(* IEC 61131-3 sources: volt/packages/volt-lsp-iec/test-corpus/lenze-mid/Device/Plc Logic/Application/Library Manager/CAA File, 66 files *)

(* ---- ATTRIB.dut ---- *)
TYPE ATTRIB :
(
	ARCHIVE := 0,
	HIDDEN,
	NORMAL,
	READONLY
);
END_TYPE

(* ---- ERROR.dut ---- *)
TYPE ERROR :
(
	NO_ERROR := 0,
	FIRST_ERROR := 5100,
	TIME_OUT,
	ABORT,
	HANDLE_INVALID,
	NOT_EXIST,
	EXIST,
	NO_MORE_ENTRIES,
	NOT_EMPTY,
	READ_ONLY_CAA,
	WRONG_PARAMETER,
	ERROR_UNKNOWN,
	WRITE_INCOMPLETE,
	FILE_NOT_IMPLEMENTED,
	ASM_CREATEJOB_FAILED,
	FILE_OPERATION_DENIED,
	FIRST_MF := 5150,
	LAST_ERROR := 5199
);
END_TYPE

(* ---- FILE_CLOSE_PARAMS.dut ---- *)
TYPE FILE_CLOSE_PARAMS :
STRUCT
	HFILE : CAA.HANDLE;
END_STRUCT
END_TYPE

(* ---- FILE_COPY_PARAMS.dut ---- *)
TYPE FILE_COPY_PARAMS :
STRUCT
	SFILENAMEDEST : CAA.FILENAME;
	SFILENAMESOURCE : CAA.FILENAME;
	XOVERWRITE : BOOL;
	ABYDUMMY : ARRAY [0..2] OF BYTE;
	SZSIZE : CAA.SIZE;
END_STRUCT
END_TYPE

(* ---- FILE_DELETE_PARAMS.dut ---- *)
TYPE FILE_DELETE_PARAMS :
STRUCT
	SFILENAME : CAA.FILENAME;
END_STRUCT
END_TYPE

(* ---- FILE_DIR_ENTRY.dut ---- *)
TYPE FILE_DIR_ENTRY :
STRUCT
	SENTRY : CAA.FILENAME;
	SZSIZE : CAA.SIZE;
	XDIRECTORY : BOOL;
	XEXCLUSIVE : BOOL;
	DTLASTMODIFICATION : DATE_AND_TIME;
END_STRUCT
END_TYPE

(* ---- FILE_DIRCLOSE_PARAMS.dut ---- *)
TYPE FILE_DIRCLOSE_PARAMS :
STRUCT
	HDIR : CAA.HANDLE;
END_STRUCT
END_TYPE

(* ---- FILE_DIRCOPY_PARAMS.dut ---- *)
TYPE FILE_DIRCOPY_PARAMS :
STRUCT
	SDIRNAMEDEST : CAA.FILENAME;
	SDIRNAMESOURCE : CAA.FILENAME;
	XRECURSIVE : BOOL;
	XOVERWRITE : BOOL;
END_STRUCT
END_TYPE

(* ---- FILE_DIRCREATE_PARAMS.dut ---- *)
TYPE FILE_DIRCREATE_PARAMS :
STRUCT
	SDIRNAME : CAA.FILENAME;
	XPARENT : BOOL;
END_STRUCT
END_TYPE

(* ---- FILE_DIRLIST_PARAMS.dut ---- *)
TYPE FILE_DIRLIST_PARAMS :
STRUCT
	HDIR : CAA.HANDLE;
	DEDIRENTRY : FILE_DIR_ENTRY;
END_STRUCT
END_TYPE

(* ---- FILE_DIROPEN_PARAMS.dut ---- *)
TYPE FILE_DIROPEN_PARAMS :
STRUCT
	SDIRNAME : CAA.FILENAME;
	HDIR : CAA.HANDLE;
END_STRUCT
END_TYPE

(* ---- FILE_DIRREMOVE_PARAMS.dut ---- *)
TYPE FILE_DIRREMOVE_PARAMS :
STRUCT
	SDIRNAME : CAA.FILENAME;
	XRECURSIVE : BOOL;
END_STRUCT
END_TYPE

(* ---- FILE_DIRRENAME_PARAMS.dut ---- *)
TYPE FILE_DIRRENAME_PARAMS :
STRUCT
	SDIRNAMEOLD : CAA.FILENAME;
	SDIRNAMENEW : CAA.FILENAME;
END_STRUCT
END_TYPE

(* ---- FILE_EOF_PARAMS.dut ---- *)
TYPE FILE_EOF_PARAMS :
STRUCT
	HFILE : CAA.HANDLE;
	XEOF : BOOL;
END_STRUCT
END_TYPE

(* ---- FILE_FLUSH_PARAMS.dut ---- *)
TYPE FILE_FLUSH_PARAMS :
STRUCT
	HFILE : CAA.HANDLE;
END_STRUCT
END_TYPE

(* ---- FILE_GETAT_PARAMS.dut ---- *)
TYPE FILE_GETAT_PARAMS :
STRUCT
	HFILE : CAA.HANDLE;
	EFILEATTRIB : ATTRIB;
END_STRUCT
END_TYPE

(* ---- FILE_GETPOS_PARAMS.dut ---- *)
TYPE FILE_GETPOS_PARAMS :
STRUCT
	HFILE : CAA.HANDLE;
	UDIPOS : __UXINT;
END_STRUCT
END_TYPE

(* ---- FILE_GETROOT_PARAMS.dut ---- *)
TYPE FILE_GETROOT_PARAMS :
STRUCT
	SFILENAME : CAA.FILENAME;
END_STRUCT
END_TYPE

(* ---- FILE_GETSIZE_PARAMS.dut ---- *)
TYPE FILE_GETSIZE_PARAMS :
STRUCT
	SFILENAME : CAA.FILENAME;
	SZSIZE : CAA.SIZE;
END_STRUCT
END_TYPE

(* ---- FILE_GETTIME_PARAMS.dut ---- *)
TYPE FILE_GETTIME_PARAMS :
STRUCT
	SFILENAME : CAA.FILENAME;
	DTLASTMODIFICATION : DATE_AND_TIME;
END_STRUCT
END_TYPE

(* ---- FILE_OPEN_PARAMS.dut ---- *)
TYPE FILE_OPEN_PARAMS :
STRUCT
	SFILENAME : CAA.FILENAME;
	EFILEMODE : MODE;
	XEXCLUSIVE : BOOL;
	BYDUMMY : BOOL;
	HFILE : CAA.HANDLE;
END_STRUCT
END_TYPE

(* ---- FILE_READ_PARAMS.dut ---- *)
TYPE FILE_READ_PARAMS :
STRUCT
	HFILE : CAA.HANDLE;
	PBUFFER : CAA.PVOID;
	SZBUFFER : CAA.SIZE;
	SZSIZE : CAA.SIZE;
END_STRUCT
END_TYPE

(* ---- FILE_RENAME_PARAMS.dut ---- *)
TYPE FILE_RENAME_PARAMS :
STRUCT
	SFILENAMEOLD : CAA.FILENAME;
	SFILENAMENEW : CAA.FILENAME;
END_STRUCT
END_TYPE

(* ---- FILE_SETAT_PARAMS.dut ---- *)
TYPE FILE_SETAT_PARAMS :
STRUCT
	HFILE : CAA.HANDLE;
	EFILEATTRIB : ATTRIB;
END_STRUCT
END_TYPE

(* ---- FILE_SETPOS_PARAMS.dut ---- *)
TYPE FILE_SETPOS_PARAMS :
STRUCT
	HFILE : CAA.HANDLE;
	UDIPOS : __UXINT;
END_STRUCT
END_TYPE

(* ---- FILE_SETROOT_PARAMS.dut ---- *)
TYPE FILE_SETROOT_PARAMS :
STRUCT
	SFILENAME : CAA.FILENAME;
END_STRUCT
END_TYPE

(* ---- FILE_WRITE_PARAMS.dut ---- *)
TYPE FILE_WRITE_PARAMS :
STRUCT
	HFILE : CAA.HANDLE;
	PBUFFER : CAA.PVOID;
	SZSIZE : CAA.SIZE;
END_STRUCT
END_TYPE

(* ---- MODE.dut ---- *)
TYPE MODE :
(
	MWRITE := 0,
	MREAD,
	MRDWR,
	MAPPD,
	MREADPLUS,
	MWRITEPLUS,
	MAPPENDPLUS
);
END_TYPE

(* ---- CAA_ASM_CONSTANTS.gvl ---- *)
VAR_GLOBAL
	OPEN_JOB_ID : UDINT := 16#10001;
	CLOSE_JOB_ID : UDINT := 16#10002;
	COPY_JOB_ID : UDINT := 16#10003;
	DELETE_JOB_ID : UDINT := 16#10004;
	EOF_JOB_ID : UDINT := 16#10005;
	GETPOS_JOB_ID : UDINT := 16#10006;
	GETSIZE_JOB_ID : UDINT := 16#10007;
	GETTIME_JOB_ID : UDINT := 16#10008;
	READ_JOB_ID : UDINT := 16#10009;
	RENAME_JOB_ID : UDINT := 16#1000A;
	SETATTRIBUTE_JOB_ID : UDINT := 16#1000B;
	SETPOS_JOB_ID : UDINT := 16#1000C;
	WRITE_JOB_ID : UDINT := 16#1000D;
	GETROOT_JOB_ID : UDINT := 16#1000E;
	SETROOT_JOB_ID : UDINT := 16#1000F;
	DIRCLOSE_JOB_ID : UDINT := 16#10010;
	DIRCREATE_JOB_ID : UDINT := 16#10011;
	DIRLIST_JOB_ID : UDINT := 16#10012;
	DIROPEN_JOB_ID : UDINT := 16#10013;
	DIRREMOVE_JOB_ID : UDINT := 16#10014;
	DIRRENAME_JOB_ID : UDINT := 16#10015;
	FLUSH_JOB_ID : UDINT := 16#10016;
	GETATTRIBUTE_JOB_ID : UDINT := 16#10017;
	DIRCOPY_JOB_ID : UDINT := 16#10018;
END_VAR

(* ---- CAA_GLOBALE_CONSTANTS.gvl ---- *)
VAR_GLOBAL
	GC_PDIRNAME : WORD := 1;
	GC_PRENAME : WORD := 2;
	GC_PCOPY : WORD := 3;
	GC_PSETATTRIBUTE : WORD := 4;
	GC_PFILENAME83 : WORD := 100;
	GC_PCAPITALLETTERS : WORD := 101;
	GC_PABSOLUTEPATH : WORD := 200;
	GC_PDRIVELETTER : WORD := 201;
	GC_PNETWORKDRIVES : WORD := 300;
END_VAR

(* ---- EXAMPLES.gvl ---- *)
VAR_GLOBAL
	IDUMMYFORLIBDOCUCAAFILE : INT := 99;
END_VAR

(* ---- RSHANDLING.gvl ---- *)
VAR_GLOBAL
	G_FILECLASS : FileClass;
	G_DIRCLASS : DirClass;
END_VAR

(* ---- VERSIONCONSTANTS.gvl ---- *)
VAR_GLOBAL
	GC_BYVERSION : BYTE := 1;
	GC_BYVERSION_1 : BYTE := 0;
END_VAR

(* ---- _CLOSE.pou ---- *)
FUNCTION _CLOSE : ERROR
VAR_INPUT
	HFILE : CAA.HANDLE;
END_VAR
END_FUNCTION

(* ---- _DIRCLOSE.pou ---- *)
FUNCTION _DIRCLOSE : ERROR
VAR_INPUT
	HDIR : CAA.HANDLE;
END_VAR
END_FUNCTION

(* ---- GETLIBVERSION.pou ---- *)
FUNCTION GETLIBVERSION : VERSION
END_FUNCTION

(* ---- GETLIBVERSIONNUMBER.pou ---- *)
FUNCTION GETLIBVERSIONNUMBER : DWORD
END_FUNCTION

(* ---- GETPROPERTY.pou ---- *)
FUNCTION GETPROPERTY : DWORD
VAR_INPUT
	WPROPERTY : WORD;
END_VAR
END_FUNCTION

(* ---- GETSUPPLIERVERSION.pou ---- *)
FUNCTION GETSUPPLIERVERSION : WORD
VAR_INPUT
	XDUMMY : BOOL;
END_VAR
END_FUNCTION

(* ---- ISLIBRELEASED.pou ---- *)
FUNCTION ISLIBRELEASED : BOOL
END_FUNCTION

(* ---- CLOSE.pou ---- *)
FUNCTION_BLOCK CLOSE EXTENDS ETrig
VAR_INPUT
	HFILE : CAA.HANDLE;
END_VAR
VAR_OUTPUT
	EERROR : ERROR;
END_VAR
VAR
	HJOB : CAA.HANDLE;
	PFILECLOSEPARAMS : POINTER TO FILE_CLOSE_PARAMS;
	STATEJOB : ASM.STATE;
	FILECLOSEPARAMS : FILE_CLOSE_PARAMS;
END_VAR
END_FUNCTION_BLOCK

METHOD PRVABORT : BOOL
END_METHOD

METHOD PRVCYCLICACTION : BOOL
END_METHOD

METHOD PRVRESETOUTPUTS : BOOL
END_METHOD

METHOD PRVSTART : BOOL
END_METHOD

(* ---- COPY.pou ---- *)
FUNCTION_BLOCK COPY EXTENDS ETrigToA
VAR_INPUT
	SFILENAMEDEST : CAA.FILENAME;
	SFILENAMESOURCE : CAA.FILENAME;
	XOVERWRITE : BOOL := TRUE;
END_VAR
VAR_OUTPUT
	EERROR : ERROR;
	SZSIZE : CAA.SIZE;
END_VAR
VAR
	HJOB : CAA.HANDLE;
	PFILECOPYPARAMS : POINTER TO FILE_COPY_PARAMS;
	STATEJOB : ASM.STATE;
	FILECOPYPARAMS : FILE_COPY_PARAMS;
END_VAR
END_FUNCTION_BLOCK

METHOD PRVABORT : BOOL
END_METHOD

METHOD PRVCYCLICACTION : BOOL
END_METHOD

METHOD PRVRESETOUTPUTS : BOOL
END_METHOD

METHOD PRVSTART : BOOL
END_METHOD

(* ---- DELETE.pou ---- *)
FUNCTION_BLOCK DELETE EXTENDS ETrig
VAR_INPUT
	SFILENAME : CAA.FILENAME;
END_VAR
VAR_OUTPUT
	EERROR : ERROR;
END_VAR
VAR
	HJOB : CAA.HANDLE;
	PFILEDELETEPARAMS : POINTER TO FILE_DELETE_PARAMS;
	STATEJOB : ASM.STATE;
	FILEDELETEPARAMS : FILE_DELETE_PARAMS;
END_VAR
END_FUNCTION_BLOCK

METHOD PRVABORT : BOOL
END_METHOD

METHOD PRVCYCLICACTION : BOOL
END_METHOD

METHOD PRVRESETOUTPUTS : BOOL
END_METHOD

METHOD PRVSTART : BOOL
END_METHOD

(* ---- DIRCLASS.pou ---- *)
FUNCTION_BLOCK DIRCLASS EXTENDS RSMClass
END_FUNCTION_BLOCK

METHOD CLOSE : RSM.ERROR
VAR_INPUT
	HHANDLE : CAA.HANDLE;
END_VAR
END_METHOD

(* ---- DIRCLOSE.pou ---- *)
FUNCTION_BLOCK DIRCLOSE EXTENDS ETrig
VAR_INPUT
	HDIR : CAA.HANDLE;
END_VAR
VAR_OUTPUT
	EERROR : ERROR;
END_VAR
VAR
	HJOB : CAA.HANDLE;
	PDIRCLOSEPARAMS : POINTER TO FILE_DIRCLOSE_PARAMS;
	STATEJOB : ASM.STATE;
	DIRCLOSEPARAMS : FILE_DIRCLOSE_PARAMS;
END_VAR
END_FUNCTION_BLOCK

METHOD PRVSTART : BOOL
END_METHOD

METHOD PRVCYCLICACTION : BOOL
END_METHOD

METHOD PRVRESETOUTPUTS : BOOL
END_METHOD

METHOD PRVABORT : BOOL
END_METHOD

(* ---- DIRCOPY.pou ---- *)
FUNCTION_BLOCK DIRCOPY EXTENDS ETrig
VAR_INPUT
	SDIRNAMEDEST : CAA.FILENAME;
	SDIRNAMESOURCE : CAA.FILENAME;
	XRECURSIVE : BOOL;
	XOVERWRITE : BOOL;
END_VAR
VAR_OUTPUT
	EERROR : ERROR;
END_VAR
VAR
	HJOB : CAA.HANDLE;
	PDIRCOPYPARAMS : POINTER TO FILE_DIRCOPY_PARAMS;
	STATEJOB : ASM.STATE;
	DIRCOPYPARAMS : FILE_DIRCOPY_PARAMS;
END_VAR
END_FUNCTION_BLOCK

METHOD PRVCYCLICACTION : BOOL
END_METHOD

METHOD PRVRESETOUTPUTS : BOOL
END_METHOD

METHOD PRVABORT : BOOL
END_METHOD

METHOD PRVSTART : BOOL
END_METHOD

(* ---- DIRCREATE.pou ---- *)
FUNCTION_BLOCK DIRCREATE EXTENDS ETrig
VAR_INPUT
	SDIRNAME : CAA.FILENAME;
	XPARENT : BOOL;
END_VAR
VAR_OUTPUT
	EERROR : ERROR;
END_VAR
VAR
	HJOB : CAA.HANDLE;
	PDIRCREATEPARAMS : POINTER TO FILE_DIRCREATE_PARAMS;
	STATEJOB : ASM.STATE;
	DIRCREATEPARAMS : FILE_DIRCREATE_PARAMS;
END_VAR
END_FUNCTION_BLOCK

METHOD PRVSTART : BOOL
END_METHOD

METHOD PRVCYCLICACTION : BOOL
END_METHOD

METHOD PRVRESETOUTPUTS : BOOL
END_METHOD

METHOD PRVABORT : BOOL
END_METHOD

(* ---- DIRLIST.pou ---- *)
FUNCTION_BLOCK DIRLIST EXTENDS ETrig
VAR_INPUT
	HDIR : CAA.HANDLE;
END_VAR
VAR_OUTPUT
	EERROR : ERROR;
	DEDIRENTRY : FILE_DIR_ENTRY;
END_VAR
VAR
	HJOB : CAA.HANDLE;
	PDIRLISTPARAMS : POINTER TO FILE_DIRLIST_PARAMS;
	STATEJOB : ASM.STATE;
	DIRLISTPARAMS : FILE_DIRLIST_PARAMS;
END_VAR
END_FUNCTION_BLOCK

METHOD PRVCYCLICACTION : BOOL
END_METHOD

METHOD PRVRESETOUTPUTS : BOOL
END_METHOD

METHOD PRVABORT : BOOL
END_METHOD

METHOD PRVSTART : BOOL
END_METHOD

(* ---- DIROPEN.pou ---- *)
FUNCTION_BLOCK DIROPEN EXTENDS ETrig
VAR_INPUT
	SDIRNAME : CAA.FILENAME;
END_VAR
VAR_OUTPUT
	EERROR : ERROR;
	HDIR : CAA.HANDLE;
END_VAR
VAR
	SCOPYDIRNAME : CAA.FILENAME;
	HJOB : CAA.HANDLE;
	PDIROPENPARAMS : POINTER TO FILE_DIROPEN_PARAMS;
	STATEJOB : ASM.STATE;
	DIROPENPARAMS : FILE_DIROPEN_PARAMS;
END_VAR
END_FUNCTION_BLOCK

METHOD PRVCYCLICACTION : BOOL
END_METHOD

METHOD PRVRESETOUTPUTS : BOOL
END_METHOD

METHOD PRVABORT : BOOL
END_METHOD

METHOD PRVSTART : BOOL
END_METHOD

(* ---- DIRREMOVE.pou ---- *)
FUNCTION_BLOCK DIRREMOVE EXTENDS ETrigToA
VAR_INPUT
	SDIRNAME : CAA.FILENAME;
	XRECURSIVE : BOOL;
END_VAR
VAR_OUTPUT
	EERROR : ERROR;
END_VAR
VAR
	HJOB : CAA.HANDLE;
	PDIRREMOVEPARAMS : POINTER TO FILE_DIRREMOVE_PARAMS;
	STATEJOB : ASM.STATE;
	DIRREMOVEPARAMS : FILE_DIRREMOVE_PARAMS;
END_VAR
END_FUNCTION_BLOCK

METHOD PRVRESETOUTPUTS : BOOL
END_METHOD

METHOD PRVABORT : BOOL
END_METHOD

METHOD PRVSTART : BOOL
END_METHOD

METHOD PRVCYCLICACTION : BOOL
END_METHOD

(* ---- DIRRENAME.pou ---- *)
FUNCTION_BLOCK DIRRENAME EXTENDS ETrig
VAR_INPUT
	SDIRNAMEOLD : CAA.FILENAME;
	SDIRNAMENEW : CAA.FILENAME;
END_VAR
VAR_OUTPUT
	EERROR : ERROR;
END_VAR
VAR
	HJOB : CAA.HANDLE;
	PDIRRENAMEPARAMS : POINTER TO FILE_DIRRENAME_PARAMS;
	STATEJOB : ASM.STATE;
	DIRRENAMEPARAMS : FILE_DIRRENAME_PARAMS;
END_VAR
END_FUNCTION_BLOCK

METHOD PRVRESETOUTPUTS : BOOL
END_METHOD

METHOD PRVABORT : BOOL
END_METHOD

METHOD PRVSTART : BOOL
END_METHOD

METHOD PRVCYCLICACTION : BOOL
END_METHOD

(* ---- EOF.pou ---- *)
FUNCTION_BLOCK EOF EXTENDS ETrig
VAR_INPUT
	HFILE : CAA.HANDLE;
END_VAR
VAR_OUTPUT
	EERROR : ERROR;
	XEOF : BOOL;
END_VAR
VAR
	HJOB : CAA.HANDLE;
	PEOFPARAMS : POINTER TO FILE_EOF_PARAMS;
	STATEJOB : ASM.STATE;
	EOFPARAMS : FILE_EOF_PARAMS;
END_VAR
END_FUNCTION_BLOCK

METHOD PRVABORT : BOOL
END_METHOD

METHOD PRVCYCLICACTION : BOOL
END_METHOD

METHOD PRVRESETOUTPUTS : BOOL
END_METHOD

METHOD PRVSTART : BOOL
END_METHOD

(* ---- FILECLASS.pou ---- *)
FUNCTION_BLOCK FILECLASS EXTENDS RSMClass
END_FUNCTION_BLOCK

METHOD CLOSE : RSM.ERROR
VAR_INPUT
	HHANDLE : CAA.HANDLE;
END_VAR
END_METHOD

(* ---- FLUSH.pou ---- *)
FUNCTION_BLOCK FLUSH EXTENDS ETrig
VAR_INPUT
	HFILE : CAA.HANDLE;
END_VAR
VAR_OUTPUT
	EERROR : ERROR;
END_VAR
VAR
	HJOB : CAA.HANDLE;
	PFLUSHPARAMS : POINTER TO FILE_FLUSH_PARAMS;
	STATEJOB : ASM.STATE;
	FLUSHPARAMS : FILE_FLUSH_PARAMS;
END_VAR
END_FUNCTION_BLOCK

METHOD PRVABORT : BOOL
END_METHOD

METHOD PRVCYCLICACTION : BOOL
END_METHOD

METHOD PRVRESETOUTPUTS : BOOL
END_METHOD

METHOD PRVSTART : BOOL
END_METHOD

(* ---- GETATTRIBUTE.pou ---- *)
FUNCTION_BLOCK GETATTRIBUTE EXTENDS ETrig
VAR_INPUT
	HFILE : CAA.HANDLE;
END_VAR
VAR_OUTPUT
	EERROR : ERROR;
	EFILEATTRIB : ATTRIB;
END_VAR
VAR
	HJOB : CAA.HANDLE;
	PGETATPARAMS : POINTER TO FILE_GETAT_PARAMS;
	STATEJOB : ASM.STATE;
	GETATPARAMS : FILE_GETAT_PARAMS;
END_VAR
END_FUNCTION_BLOCK

METHOD PRVABORT : BOOL
END_METHOD

METHOD PRVCYCLICACTION : BOOL
END_METHOD

METHOD PRVRESETOUTPUTS : BOOL
END_METHOD

METHOD PRVSTART : BOOL
END_METHOD

(* ---- GETPOS.pou ---- *)
FUNCTION_BLOCK GETPOS EXTENDS ETrig
VAR_INPUT
	HFILE : CAA.HANDLE;
END_VAR
VAR_OUTPUT
	EERROR : ERROR;
	UDIPOS : __UXINT;
END_VAR
VAR
	HJOB : CAA.HANDLE;
	PGETPOSPARAMS : POINTER TO FILE_GETPOS_PARAMS;
	STATEJOB : ASM.STATE;
	GETPOSPARAMS : FILE_GETPOS_PARAMS;
END_VAR
END_FUNCTION_BLOCK

METHOD PRVABORT : BOOL
END_METHOD

METHOD PRVCYCLICACTION : BOOL
END_METHOD

METHOD PRVRESETOUTPUTS : BOOL
END_METHOD

METHOD PRVSTART : BOOL
END_METHOD

(* ---- GETROOT.pou ---- *)
FUNCTION_BLOCK GETROOT EXTENDS ETrig
VAR_OUTPUT
	EERROR : ERROR;
	SFILENAME : CAA.FILENAME;
END_VAR
VAR
	HJOB : CAA.HANDLE;
	PGETROOTPARAMS : POINTER TO FILE_GETROOT_PARAMS;
	STATEJOB : ASM.STATE;
	GETROOTPARAMS : FILE_GETROOT_PARAMS;
END_VAR
END_FUNCTION_BLOCK

METHOD PRVCYCLICACTION : BOOL
END_METHOD

METHOD PRVRESETOUTPUTS : BOOL
END_METHOD

METHOD PRVABORT : BOOL
END_METHOD

METHOD PRVSTART : BOOL
END_METHOD

(* ---- GETSIZE.pou ---- *)
FUNCTION_BLOCK GETSIZE EXTENDS ETrig
VAR_INPUT
	SFILENAME : CAA.FILENAME;
END_VAR
VAR_OUTPUT
	EERROR : ERROR;
	SZSIZE : CAA.SIZE;
END_VAR
VAR
	HJOB : CAA.HANDLE;
	PGETSIZEPARAMS : POINTER TO FILE_GETSIZE_PARAMS;
	STATEJOB : ASM.STATE;
	GETSIZEPARAMS : FILE_GETSIZE_PARAMS;
END_VAR
END_FUNCTION_BLOCK

METHOD PRVABORT : BOOL
END_METHOD

METHOD PRVCYCLICACTION : BOOL
END_METHOD

METHOD PRVRESETOUTPUTS : BOOL
END_METHOD

METHOD PRVSTART : BOOL
END_METHOD

(* ---- GETTIME.pou ---- *)
FUNCTION_BLOCK GETTIME EXTENDS ETrig
VAR_INPUT
	SFILENAME : CAA.FILENAME;
END_VAR
VAR_OUTPUT
	EERROR : ERROR;
	DTLASTMODIFICATION : DATE_AND_TIME;
END_VAR
VAR
	HJOB : CAA.HANDLE;
	PGETTIMEPARAMS : POINTER TO FILE_GETTIME_PARAMS;
	STATEJOB : ASM.STATE;
	GETTIMEPARAMS : FILE_GETTIME_PARAMS;
END_VAR
END_FUNCTION_BLOCK

METHOD PRVABORT : BOOL
END_METHOD

METHOD PRVCYCLICACTION : BOOL
END_METHOD

METHOD PRVRESETOUTPUTS : BOOL
END_METHOD

METHOD PRVSTART : BOOL
END_METHOD

(* ---- OPEN.pou ---- *)
FUNCTION_BLOCK OPEN EXTENDS ETrig
VAR_INPUT
	SFILENAME : CAA.FILENAME;
	EFILEMODE : MODE;
	XEXCLUSIVE : BOOL;
END_VAR
VAR_OUTPUT
	EERROR : ERROR;
	HFILE : CAA.HANDLE;
END_VAR
VAR
	HJOB : CAA.HANDLE;
	PFILEOPENPARAMS : POINTER TO FILE_OPEN_PARAMS;
	STATEJOB : ASM.STATE;
	FILEOPENPARAMS : FILE_OPEN_PARAMS;
END_VAR
END_FUNCTION_BLOCK

METHOD PRVABORT : BOOL
END_METHOD

METHOD PRVCYCLICACTION : BOOL
END_METHOD

METHOD PRVRESETOUTPUTS : BOOL
END_METHOD

METHOD PRVSTART : BOOL
END_METHOD

(* ---- READ.pou ---- *)
FUNCTION_BLOCK READ EXTENDS ETrigToA
VAR_INPUT
	HFILE : CAA.HANDLE;
	PBUFFER : CAA.PVOID;
	SZBUFFER : CAA.SIZE;
END_VAR
VAR_OUTPUT
	EERROR : ERROR;
	SZSIZE : CAA.SIZE;
END_VAR
VAR
	HJOB : CAA.HANDLE;
	PREADPARAMS : POINTER TO FILE_READ_PARAMS;
	STATEJOB : ASM.STATE;
	READPARAMS : FILE_READ_PARAMS;
END_VAR
END_FUNCTION_BLOCK

METHOD PRVABORT : BOOL
END_METHOD

METHOD PRVCYCLICACTION : BOOL
END_METHOD

METHOD PRVRESETOUTPUTS : BOOL
END_METHOD

METHOD PRVSTART : BOOL
END_METHOD

(* ---- RENAME.pou ---- *)
FUNCTION_BLOCK RENAME EXTENDS ETrig
VAR_INPUT
	SFILENAMEOLD : CAA.FILENAME;
	SFILENAMENEW : CAA.FILENAME;
END_VAR
VAR_OUTPUT
	EERROR : ERROR;
END_VAR
VAR
	HJOB : CAA.HANDLE;
	PRENAMEPARAMS : POINTER TO FILE_RENAME_PARAMS;
	STATEJOB : ASM.STATE;
	RENAMEPARAMS : FILE_RENAME_PARAMS;
END_VAR
END_FUNCTION_BLOCK

METHOD PRVABORT : BOOL
END_METHOD

METHOD PRVCYCLICACTION : BOOL
END_METHOD

METHOD PRVRESETOUTPUTS : BOOL
END_METHOD

METHOD PRVSTART : BOOL
END_METHOD

(* ---- SETATTRIBUTE.pou ---- *)
FUNCTION_BLOCK SETATTRIBUTE EXTENDS ETrig
VAR_INPUT
	HFILE : CAA.HANDLE;
	EFILEATTRIB : ATTRIB;
END_VAR
VAR_OUTPUT
	EERROR : ERROR;
END_VAR
VAR
	HJOB : CAA.HANDLE;
	PSETATPARAMS : POINTER TO FILE_SETAT_PARAMS;
	STATEJOB : ASM.STATE;
	SETATPARAMS : FILE_SETAT_PARAMS;
END_VAR
END_FUNCTION_BLOCK

METHOD PRVABORT : BOOL
END_METHOD

METHOD PRVCYCLICACTION : BOOL
END_METHOD

METHOD PRVRESETOUTPUTS : BOOL
END_METHOD

METHOD PRVSTART : BOOL
END_METHOD

(* ---- SETPOS.pou ---- *)
FUNCTION_BLOCK SETPOS EXTENDS ETrig
VAR_INPUT
	HFILE : CAA.HANDLE;
	UDIPOS : __UXINT;
END_VAR
VAR_OUTPUT
	EERROR : ERROR;
END_VAR
VAR
	HJOB : CAA.HANDLE;
	PSETPOSPARAMS : POINTER TO FILE_SETPOS_PARAMS;
	STATEJOB : ASM.STATE;
	SETPOSPARAMS : FILE_SETPOS_PARAMS;
END_VAR
END_FUNCTION_BLOCK

METHOD PRVABORT : BOOL
END_METHOD

METHOD PRVCYCLICACTION : BOOL
END_METHOD

METHOD PRVRESETOUTPUTS : BOOL
END_METHOD

METHOD PRVSTART : BOOL
END_METHOD

(* ---- SETROOT.pou ---- *)
FUNCTION_BLOCK SETROOT EXTENDS ETrig
VAR_INPUT
	SFILENAME : CAA.FILENAME;
END_VAR
VAR_OUTPUT
	EERROR : ERROR;
END_VAR
VAR
	HJOB : CAA.HANDLE;
	PSETROOTPARAMS : POINTER TO FILE_SETROOT_PARAMS;
	STATEJOB : ASM.STATE;
	SETROOTPARAMS : FILE_SETROOT_PARAMS;
END_VAR
END_FUNCTION_BLOCK

METHOD PRVABORT : BOOL
END_METHOD

METHOD PRVSTART : BOOL
END_METHOD

METHOD PRVCYCLICACTION : BOOL
END_METHOD

METHOD PRVRESETOUTPUTS : BOOL
END_METHOD

(* ---- WRITE.pou ---- *)
FUNCTION_BLOCK WRITE EXTENDS ETrigToA
VAR_INPUT
	HFILE : CAA.HANDLE;
	PBUFFER : CAA.PVOID;
	SZSIZE : CAA.SIZE;
END_VAR
VAR_OUTPUT
	EERROR : ERROR;
END_VAR
VAR
	HJOB : CAA.HANDLE;
	PWRITEPARAMS : POINTER TO FILE_WRITE_PARAMS;
	STATEJOB : ASM.STATE;
	WRITEPARAMS : FILE_WRITE_PARAMS;
END_VAR
END_FUNCTION_BLOCK

METHOD PRVABORT : BOOL
END_METHOD

METHOD PRVCYCLICACTION : BOOL
END_METHOD

METHOD PRVRESETOUTPUTS : BOOL
END_METHOD

METHOD PRVSTART : BOOL
END_METHOD
